(* IEC 61131-3 sources: digital-academy-template/src, 23 files *)

(* ---- Tipi.st ---- *)
NAMESPACE tipi

    TYPE  stato : (stop, forward, backward, unknown, error);
    END_TYPE

    TYPE
        colore : USINT (
            Undefined := USINT#0, // il pacco va nel magazzino "scarto feed"
            Red       := USINT#1,
            Orange    := USINT#2,
            Yellow    := USINT#3,
            Green     := USINT#4,
            Blue      := USINT#5,
            Indigo    := USINT#6,
            Violet    := USINT#7
        ) := Undefined;
    END_TYPE

    TYPE InventoryMode:
        (Fill, Empty);
    END_TYPE

END_NAMESPACE

(* ---- tipi.st ---- *)
NAMESPACE tipi

    TYPE  stato : (stop, forward, backward, unknown, error);
    END_TYPE

END_NAMESPACE

(* ---- function.st ---- *)
NAMESPACE Libreria

    FUNCTION  SelectSensorInput : USINT
        VAR_INPUT
            uIndex : USINT;
            in1 : USINT;
            in2 : USINT;
            in3 : USINT;
            in4 : USINT;
            in5 : USINT;
        END_VAR
        CASE uIndex OF
            USINT#0 : SelectSensorInput:= in1;
            USINT#1 : SelectSensorInput:= in2;
            USINT#2 : SelectSensorInput:= in3;
            USINT#3 : SelectSensorInput:= in4;
            USINT#4 : SelectSensorInput:= in5;
        END_CASE;
    END_FUNCTION
 END_NAMESPACE

(* ---- nonusato_function.st ---- *)
NAMESPACE Libreria

    FUNCTION  SelectSensorInput : USINT
        VAR_INPUT
            uIndex : USINT;
            in1 : USINT;
            in2 : USINT;
            in3 : USINT;
            in4 : USINT;
            in5 : USINT;
        END_VAR
        CASE uIndex OF
            USINT#0 : SelectSensorInput:= in1;
            USINT#1 : SelectSensorInput:= in2;
            USINT#2 : SelectSensorInput:= in3;
            USINT#3 : SelectSensorInput:= in4;
            USINT#4 : SelectSensorInput:= in5;
        END_CASE;
    END_FUNCTION
 END_NAMESPACE

(* ---- nonusato_Simulazione.st ---- *)
USING tipi;
USING System.Timer;
USING tempo;

NAMESPACE Libreria

    FUNCTION Simulazione

        VAR_INPUT
            Qnf : BOOL;
            Qdf : BOOL;
            Qtf : BOOL;
            Qn2 : BOOL;
            Qd2 : BOOL;
            Qt2 : BOOL;
            Qn3 : BOOL;
            Qd3 : BOOL;
            Qt3 : BOOL;
            Qn4 : BOOL;
            Qd4 : BOOL;
            Qt4 : BOOL;
            Qnc : BOOL;
            Qdc : BOOL;
            Qtc : BOOL;
        END_VAR

        VAR_OUTPUT
            Idf : USINT;
            Iff : BOOL := TRUE;
            Isf : BOOL;
            Imf : BOOL;
            Id2 : USINT;
            If2 : BOOL;
            Is2 : BOOL;
            Im2 : BOOL;
            Id3 : USINT;
            If3 : BOOL;
            Is3 : BOOL;
            Im3 : BOOL;
            Id4 : USINT;
            If4 : BOOL;
            Is4 : BOOL;
            Im4 : BOOL;
            Idc : USINT;
            Ifc : BOOL;
            Isc : BOOL;
            Imc : BOOL;
        END_VAR

        VAR_EXTERNAL
            elapsedtimer : tempo.Timer;
        END_VAR

        VAR
            tStopMotor : Time;//tempo movimento motori
        END_VAR

        //BLOCCO FEED
        IF Qnf AND Iff THEN //IF nastro principale feed va avanti AND pacco presente su nastro principale feed
            IF elapsedtimer.Check(Qnf,tStopMotor) THEN //TIMER DA SISTEMARE
                Iff := FALSE; //spegni fotocellula nastro principare feed
                Isf := TRUE; //accendi sensore pacco prima del deviatore feed
                //Idf := ... ; //il sensore riceve il colore del pacco
            END_IF;
        END_IF;

        IF Qdf AND Isf THEN //IF deviatore feed chiuso (sta deviando) AND pacco presente prima del deviatore feed
            //NB: il main attualmente non cambia i valori nel vettore Qd
            Isf := FALSE; //spegni sensore pacco prima del deviatore feed
            Imf := TRUE; //accendi fotocellula nastromagazzino feed
            IF Qtf AND elapsedtimer.Check(Imf,tStopMotor) THEN //IF nastro magazzino feed va avanti AND tempo passato
                Imf := FALSE;
            END_IF; //il pacco è arrivato al magazzino feed
        END_IF;

        //BLOCCO 2
        IF Qn2 AND If2 THEN //IF nastro principale va avanti AND pacco presente su nastro principale
            IF elapsedtimer.Check(Qnf,tStopMotor) THEN //TIMER DA SISTEMARE
                If2 := FALSE; //spegni fotocellula nastro principale
                Is2 := TRUE; //accendi sensore pacco prima del deviatore
                //Id2 := ... ; //il sensore riceve il colore del pacco
            END_IF;
        END_IF;

        IF Qd2 AND Is2 THEN //IF deviatore chiuso (sta deviando) AND pacco presente prima del deviatore
            //NB: il main attualmente non cambia i valori nel vettore Qd
            Is2 := FALSE; //spegni sensore pacco prima del deviatore
            Im2 := TRUE; //accendi fotocellula nastro magazzino
            IF Qt2 AND elapsedtimer.Check(Imf,tStopMotor) THEN //IF nastro magazzino va avanti AND tempo passato
                Im2 := FALSE;
            END_IF; //il pacco è arrivato al magazzino
        END_IF;

        //BLOCCO 3
        IF Qn3 AND If3 THEN //IF nastro principale va avanti AND pacco presente su nastro principale
            IF elapsedtimer.Check(Qnf,tStopMotor) THEN //TIMER DA SISTEMARE
                If3 := FALSE; //spegni fotocellula nastro principale
                Is3 := TRUE; //accendi sensore pacco prima del deviatore
                //Id3 := ... ; //il sensore riceve il colore del pacco
            END_IF;
        END_IF;

        IF Qd3 AND Is3 THEN //IF deviatore chiuso (sta deviando) AND pacco presente prima del deviatore
            //NB: il main attualmente non cambia i valori nel vettore Qd
            Is3 := FALSE; //spegni sensore pacco prima del deviatore
            Im3 := TRUE; //accendi fotocellula nastro magazzino feed
            IF Qt3 AND elapsedtimer.Check(Imf,tStopMotor) THEN //IF nastro magazzino va avanti AND tempo passato
                Im3 := FALSE;
            END_IF; //il pacco è arrivato al magazzino
        END_IF;

        //BLOCCO 4
        IF Qn4 AND If4 THEN //IF nastro principale va avanti AND pacco presente su nastro principale
            IF elapsedtimer.Check(Qnf,tStopMotor) THEN //TIMER DA SISTEMARE
                If4 := FALSE; //spegni fotocellula nastro principale
                Is4 := TRUE; //accendi sensore pacco prima del deviatore
                //Id4 := ... ; //il sensore riceve il colore del pacco
            END_IF;
        END_IF;

        IF Qd4 AND Is4 THEN //IF deviatore chiuso (sta deviando) AND pacco presente prima del deviatore
            //NB: il main attualmente non cambia i valori nel vettore Qd
            Is4 := FALSE; //spegni sensore pacco prima del deviatore
            Im4 := TRUE; //accendi fotocellula nastromagazzino
            IF Qt4 AND elapsedtimer.Check(Imf,tStopMotor) THEN //IF nastro magazzino va avanti AND tempo passato
                Im4 := FALSE;
            END_IF; //il pacco è arrivato al magazzino
        END_IF;

        //BLOCCO CODA
        IF Qnc AND Ifc THEN //IF nastro principale va avanti AND pacco presente su nastro principale
            IF elapsedtimer.Check(Qnf,tStopMotor) THEN //TIMER DA SISTEMARE
                Ifc := FALSE; //spegni fotocellula nastro principale
                Isc := TRUE; //accendi sensore pacco prima del deviatore
                //Idc := ... ; //il sensore riceve il colore del pacco
            END_IF;
        END_IF;

        IF Qdc AND Isc THEN //IF deviatore chiuso (sta deviando) AND pacco presente prima del deviatore
            //NB: il main attualmente non cambia i valori nel vettore Qd
            Isc := FALSE; //spegni sensore pacco prima del deviatore
            Imc := TRUE; //accendi fotocellula nastromagazzino
            IF Qtc AND elapsedtimer.Check(Imf,tStopMotor) THEN //IF nastro magazzino va avanti AND tempo passato
                Imc := FALSE;
            END_IF; //il pacco è arrivato al magazzino
        END_IF;

    END_FUNCTION

END_NAMESPACE

(* ---- SelectSensorInput.st ---- *)
NAMESPACE Libreria

    FUNCTION  SelectSensorInput : USINT
        VAR_INPUT
            uIndex : INT;
            in1 : USINT; //sensore colore deviatore nastro feed
            in2 : USINT; //sensore colore deviatore magazzino 2
            in3 : USINT; //sensore colore deviatore magazzino 3
            in4 : USINT; //sensore colore deviatore magazzino 4
            in5 : USINT; //sensore colore deviatore magazzino coda
        END_VAR
        CASE uIndex OF
            INT#1 : SelectSensorInput:= in1;
            INT#2 : SelectSensorInput:= in2;
            INT#3 : SelectSensorInput:= in3;
            INT#4 : SelectSensorInput:= in4;
            INT#5 : SelectSensorInput:= in5;
        END_CASE;
    END_FUNCTION
 END_NAMESPACE

(* ---- Simulazione.st ---- *)
//NOT WORKING PROPERLY AND NOT USED

USING tipi;
USING System.Timer;
USING tempo;

NAMESPACE Libreria

    FUNCTION Simulazione

        VAR_INPUT
            Qnf : BOOL;
            Qdf : BOOL;
            Qtf : BOOL;
            Qn2 : BOOL;
            Qd2 : BOOL;
            Qt2 : BOOL;
            Qn3 : BOOL;
            Qd3 : BOOL;
            Qt3 : BOOL;
            Qn4 : BOOL;
            Qd4 : BOOL;
            Qt4 : BOOL;
            Qnc : BOOL;
            Qdc : BOOL;
            Qtc : BOOL;
        END_VAR

        VAR_OUTPUT
            Idf : USINT;
            Iff : BOOL := TRUE;
            Isf : BOOL;
            Imf : BOOL;
            Id2 : USINT;
            If2 : BOOL;
            Is2 : BOOL;
            Im2 : BOOL;
            Id3 : USINT;
            If3 : BOOL;
            Is3 : BOOL;
            Im3 : BOOL;
            Id4 : USINT;
            If4 : BOOL;
            Is4 : BOOL;
            Im4 : BOOL;
            Idc : USINT;
            Ifc : BOOL;
            Isc : BOOL;
            Imc : BOOL;
        END_VAR

        VAR_EXTERNAL
            elapsedtimer : tempo.Timer;
        END_VAR

        VAR
            tStopMotor : Time;//tempo movimento motori
        END_VAR

        //BLOCCO FEED
        IF Qnf AND Iff THEN //IF nastro principale feed va avanti AND pacco presente su nastro principale feed
            IF elapsedtimer.Check(Qnf,tStopMotor) THEN //TIMER DA SISTEMARE
                Iff := FALSE; //spegni fotocellula nastro principare feed
                Isf := TRUE; //accendi sensore pacco prima del deviatore feed
                //Idf := ... ; //il sensore riceve il colore del pacco
            END_IF;
        END_IF;

        IF Qdf AND Isf THEN //IF deviatore feed chiuso (sta deviando) AND pacco presente prima del deviatore feed
            //NB: il main attualmente non cambia i valori nel vettore Qd
            Isf := FALSE; //spegni sensore pacco prima del deviatore feed
            Imf := TRUE; //accendi fotocellula nastromagazzino feed
            IF Qtf AND elapsedtimer.Check(Imf,tStopMotor) THEN //IF nastro magazzino feed va avanti AND tempo passato
                Imf := FALSE;
            END_IF; //il pacco è arrivato al magazzino feed
        END_IF;

        //BLOCCO 2
        IF Qn2 AND If2 THEN //IF nastro principale va avanti AND pacco presente su nastro principale
            IF elapsedtimer.Check(Qnf,tStopMotor) THEN //TIMER DA SISTEMARE
                If2 := FALSE; //spegni fotocellula nastro principale
                Is2 := TRUE; //accendi sensore pacco prima del deviatore
                //Id2 := ... ; //il sensore riceve il colore del pacco
            END_IF;
        END_IF;

        IF Qd2 AND Is2 THEN //IF deviatore chiuso (sta deviando) AND pacco presente prima del deviatore
            //NB: il main attualmente non cambia i valori nel vettore Qd
            Is2 := FALSE; //spegni sensore pacco prima del deviatore
            Im2 := TRUE; //accendi fotocellula nastro magazzino
            IF Qt2 AND elapsedtimer.Check(Imf,tStopMotor) THEN //IF nastro magazzino va avanti AND tempo passato
                Im2 := FALSE;
            END_IF; //il pacco è arrivato al magazzino
        END_IF;

        //BLOCCO 3
        IF Qn3 AND If3 THEN //IF nastro principale va avanti AND pacco presente su nastro principale
            IF elapsedtimer.Check(Qnf,tStopMotor) THEN //TIMER DA SISTEMARE
                If3 := FALSE; //spegni fotocellula nastro principale
                Is3 := TRUE; //accendi sensore pacco prima del deviatore
                //Id3 := ... ; //il sensore riceve il colore del pacco
            END_IF;
        END_IF;

        IF Qd3 AND Is3 THEN //IF deviatore chiuso (sta deviando) AND pacco presente prima del deviatore
            //NB: il main attualmente non cambia i valori nel vettore Qd
            Is3 := FALSE; //spegni sensore pacco prima del deviatore
            Im3 := TRUE; //accendi fotocellula nastro magazzino feed
            IF Qt3 AND elapsedtimer.Check(Imf,tStopMotor) THEN //IF nastro magazzino va avanti AND tempo passato
                Im3 := FALSE;
            END_IF; //il pacco è arrivato al magazzino
        END_IF;

        //BLOCCO 4
        IF Qn4 AND If4 THEN //IF nastro principale va avanti AND pacco presente su nastro principale
            IF elapsedtimer.Check(Qnf,tStopMotor) THEN //TIMER DA SISTEMARE
                If4 := FALSE; //spegni fotocellula nastro principale
                Is4 := TRUE; //accendi sensore pacco prima del deviatore
                //Id4 := ... ; //il sensore riceve il colore del pacco
            END_IF;
        END_IF;

        IF Qd4 AND Is4 THEN //IF deviatore chiuso (sta deviando) AND pacco presente prima del deviatore
            //NB: il main attualmente non cambia i valori nel vettore Qd
            Is4 := FALSE; //spegni sensore pacco prima del deviatore
            Im4 := TRUE; //accendi fotocellula nastromagazzino
            IF Qt4 AND elapsedtimer.Check(Imf,tStopMotor) THEN //IF nastro magazzino va avanti AND tempo passato
                Im4 := FALSE;
            END_IF; //il pacco è arrivato al magazzino
        END_IF;

        //BLOCCO CODA
        IF Qnc AND Ifc THEN //IF nastro principale va avanti AND pacco presente su nastro principale
            IF elapsedtimer.Check(Qnf,tStopMotor) THEN //TIMER DA SISTEMARE
                Ifc := FALSE; //spegni fotocellula nastro principale
                Isc := TRUE; //accendi sensore pacco prima del deviatore
                //Idc := ... ; //il sensore riceve il colore del pacco
            END_IF;
        END_IF;

        IF Qdc AND Isc THEN //IF deviatore chiuso (sta deviando) AND pacco presente prima del deviatore
            //NB: il main attualmente non cambia i valori nel vettore Qd
            Isc := FALSE; //spegni sensore pacco prima del deviatore
            Imc := TRUE; //accendi fotocellula nastromagazzino
            IF Qtc AND elapsedtimer.Check(Imf,tStopMotor) THEN //IF nastro magazzino va avanti AND tempo passato
                Imc := FALSE;
            END_IF; //il pacco è arrivato al magazzino
        END_IF;

    END_FUNCTION

END_NAMESPACE

(* ---- Tempo.st ---- *)
FUNCTION Timer: BOOL
    VAR_INPUT
        tStopMotor: INT;   // Tempo massimo che la funzione aspetta
    END_VAR

    VAR
        tTemp: INT := 0;   // Variabile temporanea per il conteggio
    END_VAR

    Timer:=FALSE;
    // Ciclo WHILE per incrementare il valore di t fino a tStopMotor
    WHILE tTemp < tStopMotor DO
        tTemp := tTemp + 1;
    END_WHILE;

    // Dopo aver completato il ciclo, ritorna TRUE (indica che è finito)
    Timer := TRUE;

END_FUNCTION

(* ---- Deviatore.st ---- *)
USING Tipi;

NAMESPACE Libreria

    CLASS deviatore

        VAR PUBLIC
            ID :INT;
            color : colore;
            sensore : BOOL; // il sensore del deviatore del magazzino rosso si attiva se vede un pacco rosso
            cntrlApri : BOOL; // segnale per aprire il deviatore (se è aperto lascia passare i pacchi)
            cntrlChiudi : BOOL; // segnale per chiudere il deviatore (se è chiuso devia i pacchi)
            chiuso : BOOL;
            accetta : BOOL;
        END_VAR

        METHOD PUBLIC Init // inizializzazione del deviatore
            VAR_INPUT
                IDinit : INT;
            END_VAR
            ID:=IDinit;
            sensore := FALSE; // all'inizio non vede il pacco
            chiuso := FALSE; // all'inizio il deviatore è aperto
            cntrlApri := FALSE;
            cntrlChiudi := FALSE; // all'inizio non ci sono comandi di apertura o chiusura
        END_METHOD

        METHOD PUBLIC ChiudiDeviatore : BOOL // nel main se (sensore = TRUE) vogliamo chiudere il deviatore

            cntrlChiudi := TRUE;

        END_METHOD

        METHOD PUBLIC ApriDeviatore : BOOL // una volta deviato il pacco nel mai (sensore = FALSE) vogliamo aprire il deviatore
            cntrlApri := TRUE;
            cntrlChiudi := FALSE;
            chiuso := FALSE;
        END_METHOD // NB ci pensa test.st a definire (chiuso := FALSE)

        METHOD PUBLIC Accept

            cntrlChiudi := TRUE;

        END_METHOD

        METHOD PUBLIC Discard : BOOL

            cntrlApri := TRUE;

        END_METHOD

        METHOD PUBLIC IsMyColor : BOOL  //controlla se accettare o meno il pacco
            VAR_INPUT
                uSensor:colore;
            END_VAR

            IF uSensor = color THEN
                IsMyColor := TRUE;
            ELSE
                IsMyColor := FALSE;
            END_IF;

        END_METHOD

    END_CLASS

END_NAMESPACE

(* ---- deviatore.st ---- *)
USING Tipi;

NAMESPACE Libreria

    CLASS deviatore

        VAR PUBLIC
            ID :INT;
            sensore : BOOL; // il sensore del deviatore del magazzino rosso si attiva se vede un pacco rosso
            cntrlApri : BOOL; // segnale per aprire il deviatore (se è aperto lascia passare i pacchi)
            cntrlChiudi : BOOL; // segnale per chiudere il deviatore (se è chiuso devia i pacchi)
            chiuso : BOOL;
        END_VAR

        METHOD PUBLIC Init // inizializzazione del deviatore
            VAR_INPUT
                IDinit : INT;
            END_VAR
            ID:=IDinit;
            sensore := FALSE; // all'inizio non vede il pacco
            chiuso := FALSE; // all'inizio il deviatore è aperto
            cntrlApri := FALSE;
            cntrlChiudi := FALSE; // all'inizio non ci sono comandi di apertura o chiusura
        END_METHOD

        METHOD PUBLIC ChiudiDeviatore // nel main se (sensore = TRUE) vogliamo chiudere il deviatore
            cntrlChiudi := TRUE;
            cntrlApri := FALSE;
        END_METHOD // NB ci pensa test.st a definire (chiuso := TRUE)

        METHOD PUBLIC ApriDeviatore // una volta deviato il pacco nel mai (sensore = FALSE) vogliamo aprire il deviatore
            cntrlApri := TRUE;
            cntrlChiudi := FALSE;
        END_METHOD // NB ci pensa test.st a definire (chiuso := FALSE)

    END_CLASS

END_NAMESPACE

(* ---- Inventory.st ---- *)
USING Tipi;
USING Libreria;

NAMESPACE Libreria

    CLASS PUBLIC Inventory EXTENDS nastro
        VAR PUBLIC
            IDpackage: INT;
            ListStoredPackages: ARRAY[1..100] OF USINT; //dato che un magazzino deve avere pacchi dello stesso colore, può servire per controllare che tutti i pacchi inseriti abbiano effettivamente lo stesso colore
            currentStockLevel: INT; //livello di stock attuale
            maxCapacity: INT; //capacità massima
            acceptedColor: USINT;
            StockisFull: BOOL;
            currentMode: Tipi.InventoryMode;
            statomotore: stato;
            recipe: Ricetta;
        END_VAR

        METHOD PUBLIC Init //initialization of the inventory
            VAR_INPUT
                Capacity : INT;
                Color : USINT;
                ID_i: INT;
            END_VAR
            maxCapacity := Capacity;
            acceptedColor := Color;
            IDpackage:= ID_i;
            currentStockLevel:=0; //ipotizzo che inizialmente i magazzini siano vuoti
            StockisFull := FALSE;
            currentMode := Tipi.InventoryMode#Fill; // di default vogliamo riempire i magazzini
        END_METHOD

        METHOD PUBLIC isFull  //controlla se il magazzino è pieno
            VAR_OUTPUT
                Load: BOOL; //TRUE:"ok puoi ancora riempire", FALSE:non puoi riempire
            END_VAR

            IF currentStockLevel < maxCapacity THEN
                StockisFull:= FALSE;
                Load:=TRUE;
            ELSE
                StockisFull:=TRUE;
                Load:=FALSE;
            END_IF;
        END_METHOD

        METHOD PUBLIC GetCurrentStockLevel : INT  //se chiamato, mostra il livello di riempimento attuale
            GetCurrentStockLevel:= currentStockLevel;
        END_METHOD

        METHOD PUBLIC EmptyFIFO
            VAR
                i: INT;
            END_VAR

            FOR i := 1 TO currentStockLevel - 1 DO
                ListStoredPackages[i] := ListStoredPackages[i + 1]; // Shift dei pacchi a sinistra (FIFO)
            END_FOR;
            ListStoredPackages[currentStockLevel] := TO_USINT(0); //resetto l'ultima posizione
            currentStockLevel := currentStockLevel - 1;

            IF currentStockLevel = 0 THEN
                statomotore := Tipi.stato#stop;
                currentMode:=Tipi.InventoryMode#Fill;
            END_IF;
        END_METHOD

        METHOD PUBLIC SetMode // MODALITà RIEMPIMENTO O SVUOTAMENTO, LOGICA:FIFO
            VAR_INPUT
                mode : Tipi.InventoryMode;
                //InventorySensor:BOOL;
                InventoryPhotocell: BOOL; //c'è un pacco sul nastro del magazzino?
                DiverterSensor: BOOL; //se TRUE il deviatore è chiuso e manda il pacco al magazzino
                ID_i: USINT;
            END_VAR
            currentMode := mode;
            IF currentMode= InventoryMode#Fill THEN
                IF StockisFull=FALSE AND DiverterSensor=TRUE AND statomotore=Tipi.stato#forward AND InventoryPhotocell=TRUE THEN
                    currentStockLevel:=currentStockLevel+1;
                    ListStoredPackages[currentStockLevel]:= ID_i; //salvo l'ID_i del pacco n nell'n-esima posizione dell'array
                ELSIF StockisFull=TRUE THEN
                    RETURN; //magari inserire una variabile tipo warningCode/exitflag...
                END_IF;
            ELSE // the mode is set to "empty"
                IF recipe.RecipeSatisfiable()=TRUE THEN //AND currentStockLevel > 0 THEN
                    statomotore := Tipi.stato#backward;
                    THIS.EmptyFIFO();
                END_IF;
            END_IF;
        END_METHOD

    END_CLASS

END_NAMESPACE

(* ---- inventory.st ---- *)
USING Tipi;

NAMESPACE Inventory_lib

    CLASS PUBLIC Inventory
        VAR PUBLIC
            IDpackage: INT;
            ListStoredPackages: ARRAY[1..100] OF USINT; //dato che un magazzino deve avere pacchi dello stesso colore, può servire per controllare che tutti i pacchi inseriti abbiano effettivamente lo stesso colore
            currentStockLevel: INT; //livello di stock attuale
            maxCapacity: INT; //capacità massima
            acceptedColor: USINT;
            StockisFull: BOOL;
            currentMode: Tipi.InventoryMode;
        END_VAR

        METHOD PUBLIC Init //initialization of the inventory
            VAR_INPUT
                Capacity : INT;
                Color : USINT; //oppure tipi.colore#... oppure semplicemente INT e lo legge da solo?
                ID: INT;
            END_VAR
            maxCapacity := Capacity;
            acceptedColor := Color;
            IDpackage:= ID; //anche qui sarebbe color... forse non ha senso avere sia color che ID
            currentStockLevel:=0; //ipotizzo che inizialmente i magazzini siano vuoti
            StockisFull:=FALSE;
            currentMode := Tipi.InventoryMode#Fill; // di default vogliamo riempire i magazzini
        END_METHOD

        METHOD PUBLIC isFull  //controlla se il magazzino è pieno
            VAR_OUTPUT
                StockisFull: BOOL;
                Load: BOOL; //TRUE:"ok puoi ancora riempire", FALSE:non puoi riempire
            END_VAR
            IF currentStockLevel < maxCapacity THEN
                StockisFull:= FALSE;
                Load:=TRUE;
            ELSE
                StockisFull:=TRUE;
                Load:=FALSE;
            END_IF;
        END_METHOD

        METHOD PUBLIC GetCurrentStockLevel : INT  //se chiamato, mostra il livello di riempimento attuale
            GetCurrentStockLevel:= currentStockLevel;
        END_METHOD

        METHOD PUBLIC SetMode // MODALITà RIEMPIMENTO O SVUOTAMENTO, LOGICA:FIFO
            VAR_INPUT
                mode : Tipi.InventoryMode;
                //InventorySensor:BOOL;
                InventoryPhotocell: BOOL; //c'è un pacco sul nastro del magazzino?
                DiverterSensor: BOOL; //se TRUE il deviatore è chiuso e manda il pacco al magazzino
                ID: USINT;
            END_VAR
            currentMode := mode;
            IF currentMode= InventoryMode#Fill THEN
                IF StockisFull=FALSE AND DiverterSensor=TRUE AND Tipi.stato=Tipi.stato#forward AND InventoryPhotocell=TRUE THEN
                    currentStockLevel:=currentStockLevel+1;
                    ListStoredPackages[currentStockLevel]:= ID; //salvo l'ID del pacco n nell'n-esima posizione dell'array
                ELSIF StockisFull=TRUE THEN
                    RETURN; //magari inserire una variabile tipo warningCode/exitflag...
                END_IF;
            /*ELSE // the mode is set to "empty"
                IF RecipeSatisfiable=TRUE AND Tipi.stato=backward THEN
                    currentStockLevel:=currentStockLevel-;
                END_IF*///DA COMPLETARE
            END_IF;
        END_METHOD

    END_CLASS

END_NAMESPACE

/*{Test}
METHOD PUBLIC MyTestMethod
    ; // AxUnit.Assert.Equal(y, x)
END_METHOD*/

(* ---- Magazzino.st ---- *)
USING Tipi;

NAMESPACE Libreria

    CLASS magazzino

        VAR PUBLIC
            ID:INT;
            isFull: BOOL;
            colore : colore;
            i:INT;
            spazio:INT;
            fotocellula:BOOL;
            actualState : stato;
            CntrlForward : BOOL;    // Comando avanti
            CntrlBackward : BOOL;   // Comando indietro
            isForward : BOOL;    // Uscita avanti
            isBackward : BOOL;   // Uscita indietro

        END_VAR

        METHOD PUBLIC Init  // Init motor
            VAR_INPUT
                IDinit : INT;
                Color : colore;
            END_VAR
            ID:=IDinit;
            colore := color;
            actualState := stato#stop;
            CntrlForward := FALSE;
            CntrlBackward := FALSE;
            isForward := FALSE;
            isBackward := FALSE;

        END_METHOD

        METHOD PUBLIC Update

            IF CntrlForward AND NOT CntrlBackward THEN
                actualState := stato#forward;
            ELSIF CntrlBackward AND NOT CntrlForward THEN
                actualState := stato#backward;
            ELSE
                actualState := stato#stop;
            END_IF;

            CASE actualState OF
                stato#forward:
                    isForward := TRUE;
                    isBackward := FALSE;
                stato#backward:
                    isForward := FALSE;
                    isBackward := TRUE;
                stato#stop:
                    isForward := FALSE;
                    isBackward := FALSE;
            END_CASE;
            END_METHOD

    END_CLASS

END_NAMESPACE

(* ---- magazzino.st ---- *)
USING Tipi;

NAMESPACE Libreria

    CLASS magazzino

        VAR PUBLIC
            ID:INT;
            isFull: BOOL;
            colore : colore;
            i:INT;
            spazio:INT;
            sensore:BOOL;
            actualState : stato;
            CntrlForward : BOOL;    // Comando avanti
            CntrlBackward : BOOL;   // Comando indietro
            isForward : BOOL;    // Uscita avanti
            isBackward : BOOL;   // Uscita indietro

        END_VAR

        METHOD PUBLIC Init  // Init motor
            VAR_INPUT
                IDinit : INT;
            END_VAR
            ID:=IDinit;
            colore := colore;
            actualState := stato#stop;
            CntrlForward := FALSE;
            CntrlBackward := FALSE;
            isForward := FALSE;
            isBackward := FALSE;

        END_METHOD

        METHOD PUBLIC Update

            IF CntrlForward AND NOT CntrlBackward THEN
                actualState := stato#forward;
            ELSIF CntrlBackward AND NOT CntrlForward THEN
                actualState := stato#backward;
            ELSE
                actualState := stato#stop;
            END_IF;

            CASE actualState OF
                stato#forward:
                    isForward := TRUE;
                    isBackward := FALSE;
                stato#backward:
                    isForward := FALSE;
                    isBackward := TRUE;
                stato#stop:
                    isForward := FALSE;
                    isBackward := FALSE;
            END_CASE;
            END_METHOD

    END_CLASS

END_NAMESPACE

(* ---- Nastro.st ---- *)
USING tipi;
//USING MotorClass; //preso da libreria di @sara_vecchio

NAMESPACE Libreria

    CLASS nastro

        VAR PUBLIC
            ID:INT;
            actualState : stato;    // Comando avanti
            CntrlBackward : BOOL;   // Comando indietro
            isForward : BOOL;    // Uscita avanti //necessario?
            isBackward : BOOL;   // Uscita indietro //necessario?
            isEmpty:BOOL;
            CntrlForward : BOOL;
            colore: colore;
        END_VAR

        METHOD PUBLIC Init  // Initialization motor
            VAR_INPUT
                IDinit : INT;
                Color : colore;
            END_VAR
            ID:=IDinit;
            colore := color;
            actualState := stato#stop;
            CntrlForward := FALSE;
            CntrlBackward := FALSE;
            isForward := FALSE;
            isBackward := FALSE;

        END_METHOD

        METHOD PUBLIC Update : stato

            IF CntrlForward AND NOT CntrlBackward THEN
                actualState := stato#forward;
            ELSIF CntrlBackward AND NOT CntrlForward THEN
                actualState := stato#backward;
            ELSE
                actualState := stato#stop;
            END_IF;

            CASE actualState OF
                stato#forward:
                    isForward := TRUE;
                    isBackward := FALSE;
                stato#backward:
                    isForward := FALSE;
                    isBackward := TRUE;
                stato#stop:
                    isForward := FALSE;
                    isBackward := FALSE;
            END_CASE;

        END_METHOD

        METHOD PUBLIC CheckEmpty : BOOL  //check if is isEmpty from sensor

            VAR_INPUT
                bLightSensor: BOOL;
            END_VAR

            IF bLightSensor THEN
                CheckEmpty := FALSE;
            ELSIF NOT bLightSensor THEN
                CheckEmpty := TRUE;
            ELSE
                actualState := stato#error;
            END_IF;

        END_METHOD

        METHOD PUBLIC GetStatus : tipi.stato // get state of the conveyor
            GetStatus := actualState;
        END_METHOD

        METHOD PUBLIC Stop : BOOL
            CntrlForward := FALSE;
            CntrlBackward := FALSE;
            actualState := stato#stop;
            //Stop:=????
        END_METHOD

        METHOD PUBLIC RunForward : BOOL //serve chiamare anche i motori?
            IF actualState <> stato#error THEN
                //Motor.Start := TRUE;
                CntrlForward := TRUE; //aggiungi sicura per eviatre che avanti e indietro possano essere attivati contemporaneamente
                actualState := stato#forward;
            END_IF;
            RunForward:=CntrlForward;
        END_METHOD

        METHOD PUBLIC RunBackward
            IF actualState <> stato#error THEN
                //Motor.Start := TRUE;
                CntrlBackward := TRUE; //aggiungi stessa sicura di sopra
                actualState := stato#backward;
            END_IF;
        END_METHOD

    END_CLASS

END_NAMESPACE

(* ---- nastro.st ---- *)
USING Tipi;

NAMESPACE Libreria

    CLASS nastro

        VAR PUBLIC
            ID:INT;
            isEmpty: BOOL;
            actualState : stato;
            CntrlForward : BOOL;    // Comando avanti
            CntrlBackward : BOOL;   // Comando indietro
            isForward : BOOL;    // Uscita avanti
            isBackward : BOOL;   // Uscita indietro
            i:INT;
        END_VAR

        METHOD PUBLIC Init  // Init motor
            VAR_INPUT
                IDinit : INT;
            END_VAR
            ID:=IDinit;
            actualState := stato#stop;
            CntrlForward := FALSE;
            CntrlBackward := FALSE;
            isForward := FALSE;
            isBackward := FALSE;

        END_METHOD

        METHOD PUBLIC Update

            IF CntrlForward AND NOT CntrlBackward THEN
                actualState := stato#forward;
            ELSIF CntrlBackward AND NOT CntrlForward THEN
                actualState := stato#backward;
            ELSE
                actualState := stato#stop;
            END_IF;

            CASE actualState OF
                stato#forward:
                    isForward := TRUE;
                    isBackward := FALSE;
                stato#backward:
                    isForward := FALSE;
                    isBackward := TRUE;
                stato#stop:
                    isForward := FALSE;
                    isBackward := FALSE;
            END_CASE;

        END_METHOD

        METHOD PUBLIC fotocellula  //check if is isEmpty from sensor
                isEmpty := TRUE;
        END_METHOD

        METHOD PUBLIC GetStatus // get state of the conveyor
            actualState:=actualState;
        END_METHOD
    END_CLASS

END_NAMESPACE

(* ---- nonusato_Ricetta.st ---- *)
USING tipi;

NAMESPACE Libreria

    CLASS PUBLIC Ricetta

        /*STRUCT RicettaTipo
            Colore: USINT; // colore desiderato
            Quantità: INT; // numero pacchi necessari
        END_STRUCT

        VAR_GLOBAL
            Ricetta : ARRAY[1..5] OF RicettaTipo; // max 5 tipi di pacchi richiesti
        END_VAR*/

        METHOD PUBLIC RecipeSatisfiable : BOOL
            VAR
                i: INT;
                matchingColor: USINT;
                matchingQuantity: INT;
                foundCount: INT;
            END_VAR

            RecipeSatisfiable := TRUE; // assumi che sia soddisfatta, fino a prova contraria

            /*FOR i := 1 TO SIZEOF(Tipi.Ricetta) DO
                matchingColor := Tipi.Ricetta[i].Colore;
                matchingQuantity := Tipi.Ricetta[i].Quantità;

                // Verifica se il magazzino ha il colore richiesto
                IF acceptedColor = matchingColor THEN
                    IF currentStockLevel < matchingQuantity THEN
                        RecipeSatisfiable := FALSE;
                        RETURN;
                    END_IF;
                END_IF;
            END_FOR;*/

        END_METHOD

        /*METHOD PUBLIC RecipeSatisfiable:BOOL
            IF Ricetta.HowMany THEN
                RecipeSatisfiable:=TRUE;
            ELSE
                RecipeSatisfiable:=FALSE;
            END_IF;
        END_METHOD*/

    END_CLASS

END_NAMESPACE

(* ---- nonusato_Tempo.st ---- *)
USING System.Timer;

NAMESPACE tempo

    Class Timer

    VAR
        ton : OnDelay;
    END_VAR

    METHOD PUBLIC Check : BOOL
        VAR_INPUT
            signal: BOOL;
            duration : time;
            timeout : time;
        END_VAR
        ton(signal := TRUE, duration := Timeout);
        IF (ton.output) THEN
            Check := TRUE;
        ELSE
           Check := FALSE;
        END_IF;
    END_METHOD

    METHOD PUBLIC Reset
        ton(signal:= FALSE);
    END_METHOD

    END_class

END_NAMESPACE

(* ---- Ricetta.st ---- *)
//TO BE COMPLETED; NOT USED YET

USING tipi;

NAMESPACE Libreria

    CLASS PUBLIC Ricetta

        /*STRUCT RicettaTipo
            Colore: USINT; // colore desiderato
            Quantità: INT; // numero pacchi necessari
        END_STRUCT

        VAR_GLOBAL
            Ricetta : ARRAY[1..5] OF RicettaTipo; // max 5 tipi di pacchi richiesti
        END_VAR*/

        METHOD PUBLIC RecipeSatisfiable : BOOL
            VAR
                i: INT;
                matchingColor: USINT;
                matchingQuantity: INT;
                foundCount: INT;
            END_VAR

            RecipeSatisfiable := TRUE; // assumi che sia soddisfatta, fino a prova contraria

            /*FOR i := 1 TO SIZEOF(Tipi.Ricetta) DO
                matchingColor := Tipi.Ricetta[i].Colore;
                matchingQuantity := Tipi.Ricetta[i].Quantità;

                // Verifica se il magazzino ha il colore richiesto
                IF acceptedColor = matchingColor THEN
                    IF currentStockLevel < matchingQuantity THEN
                        RecipeSatisfiable := FALSE;
                        RETURN;
                    END_IF;
                END_IF;
            END_FOR;*/

        END_METHOD

        /*METHOD PUBLIC RecipeSatisfiable:BOOL
            IF Ricetta.HowMany THEN
                RecipeSatisfiable:=TRUE;
            ELSE
                RecipeSatisfiable:=FALSE;
            END_IF;
        END_METHOD*/

    END_CLASS

END_NAMESPACE

(* ---- Configuration.st ---- *)
USING Siemens.Simatic.S71500.Tasks;
USING tipi;
USING Libreria;

CONFIGURATION MyConfig

    TASK Load: Startup;
    TASK Main(Interval := T#100ms,PRIORITY:=1); //di default è 50ms (minimo)

    PROGRAM P0 WITH Load: LoadConfiguration;
    PROGRAM P1 WITH Main: MainProgram;

    // Configuring IO tags
    VAR_GLOBAL

        //input output feed
        Qnf AT %Q0.0 : BOOL; //output nastro feed
        Qnc AT %Q0.1 : BOOL;
        Qn2 AT %Q0.2 : BOOL;
        Qn3 AT %Q0.3 : BOOL;
        Qn4 AT %Q0.4 : BOOL;

        Qdf AT %Q1.0 : BOOL; //output deviatore feed
        Qdc AT %Q1.1 : BOOL;
        Qd2 AT %Q1.2 : BOOL;
        Qd3 AT %Q1.3 : BOOL;
        Qd4 AT %Q1.4 : BOOL;

        Qtf AT %Q2.0 : BOOL; //output tank feed
        Qtc AT %Q2.1 : BOOL;
        Qt2 AT %Q2.2 : BOOL;
        Qt3 AT %Q2.3 : BOOL;
        Qt4 AT %Q2.4 : BOOL;

        Idf AT %IB6 : USINT; //input deviatore feed (colore)
        Idc AT %IB7 : USINT;
        Id2 AT %IB8 : USINT;
        Id3 AT %IB9 : USINT;
        Id4 AT %IB10 : USINT;

        Iff AT %I0.0 : BOOL; //input fotocellula feed (presenza pacco su nastro principale)
        Ifc AT %I0.1 : BOOL;
        If2 AT %I0.2 : BOOL;
        If3 AT %I0.3 : BOOL;
        If4 AT %I0.4 : BOOL;

        Isf AT %I1.0 : BOOL; //input sensore feed (presenza pacco su nastro principale prima del deviatore)
        Isc AT %I1.1 : BOOL;
        Is2 AT %I1.2 : BOOL;
        Is3 AT %I1.3 : BOOL;
        Is4 AT %I1.4 : BOOL;

        Imf AT %I2.0 : BOOL; //input magazzino feed (presenza pacco su nastro principale)
        Imc AT %I2.1 : BOOL;
        Im2 AT %I2.2 : BOOL;
        Im3 AT %I2.3 : BOOL;
        Im4 AT %I2.4 : BOOL;

    END_VAR

    VAR_GLOBAL

        nastri : ARRAY[1..n_mag] OF nastro;
        deviatori : ARRAY[1..n_mag] OF deviatore;
        magazzini : ARRAY[1..n_mag] OF inventory;

    END_VAR

    VAR_GLOBAL CONSTANT

        n_mag : INT := 5; // numero magazzini considerando uno feed e uno scarto e il penultimo ricetta o semplice
        capacity : INT := 20; //numero pacchi che ogni magazzino può contenere

    END_VAR

END_CONFIGURATION

PROGRAM LoadConfiguration

    VAR_EXTERNAL

        nastri : ARRAY [1..n_mag] OF Libreria.nastro;
        deviatori : ARRAY [1..n_mag] OF Libreria.deviatore;
        magazzini : ARRAY [1..n_mag] OF Libreria.inventory;

        Qnf : BOOL;
        Qdf : BOOL;
        Qtf : BOOL;
        Idf : USINT;
        Iff : BOOL;
        Isf : BOOL;
        Imf : BOOL;
        Qnc : BOOL;
        Qdc : BOOL;
        Qtc : BOOL;
        Idc : USINT;
        Ifc : BOOL;
        Isc : BOOL;
        Imc : BOOL;
        Qn2 : BOOL;
        Qd2 : BOOL;
        Qt2 : BOOL;
        Id2 : USINT;
        If2 : BOOL;
        Is2 : BOOL;
        Im2 : BOOL;
        Qn3 : BOOL;
        Qd3 : BOOL;
        Qt3 : BOOL;
        Id3 : USINT;
        If3 : BOOL;
        Is3 : BOOL;
        Im3 : BOOL;
        Qn4 : BOOL;
        Qd4 : BOOL;
        Qt4 : BOOL;
        Id4 : USINT;
        If4 : BOOL;
        Is4 : BOOL;
        Im4 : BOOL;

    END_VAR

    VAR_EXTERNAL CONSTANT
        n_mag : INT;
        capacity : INT;
    END_VAR

    //inizializzo il blocco feed
    nastri[1].Init(1);
    deviatori[1].Init(1, colore#Undefined); //qua dico anche che colore il deviatore deve accettare
    magazzini[1].Init_magazzino(1, capacity);

    //inizializzo il blocco 2
    nastri[2].Init(2);
    deviatori[2].Init(2, colore#Red); //qua dico anche che colore il deviatore deve accettare
    magazzini[2].Init_magazzino(2, capacity);

    //inizializzo il blocco 3
    nastri[3].Init(3);
    deviatori[3].Init(3, colore#White); //qua dico anche che colore il deviatore deve accettare
    magazzini[3].Init_magazzino(3, capacity);

    //inizializzo il blocco 4
    nastri[4].Init(4);
    deviatori[4].Init(4, colore#Yellow); //qua dico anche che colore il deviatore deve accettare
    magazzini[4].Init_magazzino(4, capacity);

    //inizializzo il blocco coda
    nastri[n_mag].Init(n_mag);
    deviatori[n_mag].Init(n_mag, colore#Undefined); //qua dico un colore a caso ma in realtà accetta tutto (vedi method deviatore.IsMyColor_coda)
    magazzini[n_mag].Init_magazzino(n_mag, capacity);

END_PROGRAM

(* ---- configuration.st ---- *)
CONFIGURATION MyConfiguration
    TASK Main(Priority := 1);

    PROGRAM P1 WITH Main: MainProgram;

    VAR_GLOBAL
        Tag1 : INT;
        Tag3 AT %IB4 : BYTE;
    END_VAR

    VAR_GLOBAL CONSTANT
        Tag2 : BOOL := TRUE ;
    END_VAR

END_CONFIGURATION

(* ---- LoadPlantConfiguration.st ---- *)
USING tipi;

PROGRAM LoadPlantConfiguration

    VAR_TEMP
        i:INT :=0;
    END_VAR

    VAR
    coloreq : USINT;
    END_VAR

    VAR_EXTERNAL
        nastri : ARRAY [1..n_mag] OF Libreria.nastro;
        deviatori : ARRAY [1..n_mag] OF Libreria.deviatore;
        magazzini : ARRAY [1..n_mag] OF Libreria.inventory;
        //Qn : REF_TO ARRAY[1..n_mag] of BOOL ;
        //Qd : ARRAY[1..n_mag] of BOOL ;
        //Qt : ARRAY[1..n_mag] of BOOL ;
        Id : ARRAY[1..n_mag] of USINT ;
        If_ : ARRAY[1..n_mag] of BOOL ;
        Is : ARRAY[1..n_mag] of BOOL ;
        Im : ARRAY[1..n_mag] of BOOL ;

        Qn: BYTE;
        Qd: BYTE;
        Qt: BYTE;
        //Id: BYTE;
    //    If_ :BYTE;
    //    Is:BYTE;
    //    Im:BYTE;

        Qnf : BOOL;
        Qdf : BOOL;
        Qtf : BOOL;
        Idf : USINT;
        Iff : BOOL;
        Isf : BOOL;
        Imf : BOOL;
        Qnc : BOOL;
        Qdc : BOOL;
        Qtc : BOOL;
        Idc : USINT;
        Ifc : BOOL;
        Isc : BOOL;
        Imc : BOOL;
        Qn2 : BOOL;
        Qd2 : BOOL;
        Qt2 : BOOL;
        Id2 : USINT;
        If2 : BOOL;
        Is2 : BOOL;
        Im2 : BOOL;
        Qn3 : BOOL;
        Qd3 : BOOL;
        Qt3 : BOOL;
        Id3 : USINT;
        If3 : BOOL;
        Is3 : BOOL;
        Im3 : BOOL;
        Qn4 : BOOL;
        Qd4 : BOOL;
        Qt4 : BOOL;
        Id4 : USINT;
        If4 : BOOL;
        Is4 : BOOL;
        Im4 : BOOL;
        //n_pacchi : INT;
        elapsedtimer : tempo.Timer;

    END_VAR

    VAR_EXTERNAL CONSTANT
        n_mag : INT;
        capacity : INT;
        n_pacchi : INT;
    END_VAR

        /*Qn[1]  := Qnf;
        Qn[2]  := Qn2;
        Qn[3]  := Qn3;
        Qn[4]  := Qn4;
        Qn[5]  := Qnc;

        Qd[1]  := Qdf;
        Qd[2]  := Qd2;
        Qd[3]  := Qd3;
        Qd[4]  := Qd4;
        Qd[5]  := Qdc;

        Qt[1]  := Qtf;
        Qt[2]  := Qt2;
        Qt[3]  := Qt3;
        Qt[4]  := Qt4;
        Qt[5]  := Qtc;*/

        Id[1]  := Idf;
        Id[2]  := Id2;
        Id[3]  := Id3;
        Id[4]  := Id4;
        Id[5]  := Idc;

        If_[1] := Iff;
        If_[2] := If2;
        If_[3] := If3;
        If_[4] := If4;
        If_[5] := Ifc;

        Is[1] := Isf;
        Is[2] := Is2;
        Is[3] := Is3;
        Is[4] := Is4;
        Is[5] := Isc;

        Im[1] := Imf;
        Im[2] := Im2;
        Im[3] := Im3;
        Im[4] := Im4;
        Im[5] := Imc;

        //feed
        nastri[1].ID := 1;
        nastri[1].colore := USINT#0;
        nastri[1].actualState := stato#stop;
        nastri[1].CntrlForward := FALSE;
        nastri[1].CntrlBackward := FALSE;
        nastri[1].isForward := FALSE;
        nastri[1].isBackward := FALSE;

        deviatori[1].ID:=nastri[1].ID;
        deviatori[1].sensore := FALSE;
        deviatori[1].chiuso := FALSE;
        deviatori[1].cntrlApri := FALSE;
        deviatori[1].cntrlChiudi := FALSE;
        deviatori[1].color:=USINT#0; //colre magazzino feed (da aggiornare con TUTTI i colori che non sono appartenenti ad un magazzino colore)

        magazzini[1].ID:=nastri[1].ID;
        magazzini[1].acceptedColor := USINT#0; // impostare colore
        magazzini[1].actualState := stato#stop;
        magazzini[1].CntrlForward := FALSE;
        magazzini[1].CntrlBackward := FALSE;
        magazzini[1].isForward := FALSE;
        magazzini[1].isBackward := FALSE;

        magazzini[1].maxCapacity := Capacity; // impostare capacità desiderata
        magazzini[1].currentStockLevel:=0;
        magazzini[1].StockisFull := FALSE;
        magazzini[1].currentMode := Tipi.InventoryMode#Fill; // di default vogliamo riempire i magazzini

        //coda
        nastri[n_mag].ID := n_mag;
        nastri[n_mag].colore := USINT#0;
        nastri[n_mag].actualState := stato#stop;
        nastri[n_mag].CntrlForward := FALSE;
        nastri[n_mag].CntrlBackward := FALSE;
        nastri[n_mag].isForward := FALSE;
        nastri[n_mag].isBackward := FALSE;

        deviatori[n_mag].ID:=nastri[n_mag].ID;
        deviatori[n_mag].sensore := FALSE;
        deviatori[n_mag].chiuso := FALSE;
        deviatori[n_mag].cntrlApri := FALSE;
        deviatori[n_mag].cntrlChiudi := FALSE;
        deviatori[n_mag].color:=USINT#0;

        magazzini[n_mag].ID:=nastri[n_mag].ID;
        magazzini[n_mag].acceptedColor := USINT#0; // impostare colore
        magazzini[n_mag].actualState := stato#stop;
        magazzini[n_mag].CntrlForward := FALSE;
        magazzini[n_mag].CntrlBackward := FALSE;
        magazzini[n_mag].isForward := FALSE;
        magazzini[n_mag].isBackward := FALSE;

        magazzini[n_mag].maxCapacity := Capacity; // impostare capacità desiderata
        magazzini[n_mag].currentStockLevel:=0;
        magazzini[n_mag].StockisFull := FALSE;
        magazzini[n_mag].currentMode := Tipi.InventoryMode#Fill; // di default vogliamo riempire i magazzini

        //secondo
        nastri[2].ID := 2;
        nastri[2].colore := USINT#1;
        nastri[2].actualState := stato#stop;
        nastri[2].CntrlForward := FALSE;
        nastri[2].CntrlBackward := FALSE;
        nastri[2].isForward := FALSE;
        nastri[2].isBackward := FALSE;

        deviatori[2].ID:=nastri[2].ID;
        deviatori[2].sensore := FALSE;
        deviatori[2].chiuso := FALSE;
        deviatori[2].cntrlApri := FALSE;
        deviatori[2].cntrlChiudi := FALSE;
        deviatori[2].color:=USINT#1;

        magazzini[2].ID:=nastri[2].ID;
        magazzini[2].acceptedColor := USINT#1; // impostare colore
        magazzini[2].actualState := stato#stop;
        magazzini[2].CntrlForward := FALSE;
        magazzini[2].CntrlBackward := FALSE;
        magazzini[2].isForward := FALSE;
        magazzini[2].isBackward := FALSE;

        magazzini[2].maxCapacity := Capacity; // impostare capacità desiderata
        magazzini[2].currentStockLevel:=0;
        magazzini[2].StockisFull := FALSE;
        magazzini[2].currentMode := Tipi.InventoryMode#Fill; // di default vogliamo riempire i magazzini

        //terzo
        nastri[3].ID := 3;
        nastri[3].colore := USINT#2;
        nastri[3].actualState := stato#stop;
        nastri[3].CntrlForward := FALSE;
        nastri[3].CntrlBackward := FALSE;
        nastri[3].isForward := FALSE;
        nastri[3].isBackward := FALSE;

        deviatori[3].ID:=nastri[3].ID;
        deviatori[3].sensore := FALSE;
        deviatori[3].chiuso := FALSE;
        deviatori[3].cntrlApri := FALSE;
        deviatori[3].cntrlChiudi := FALSE;
        deviatori[3].color:=USINT#2;

        magazzini[3].ID:=nastri[3].ID;
        magazzini[3].acceptedColor := USINT#2; // impostare colore
        magazzini[3].actualState := stato#stop;
        magazzini[3].CntrlForward := FALSE;
        magazzini[3].CntrlBackward := FALSE;
        magazzini[3].isForward := FALSE;
        magazzini[3].isBackward := FALSE;

        magazzini[3].maxCapacity := Capacity; // impostare capacità desiderata
        magazzini[3].currentStockLevel:=0;
        magazzini[3].StockisFull := FALSE;
        magazzini[3].currentMode := Tipi.InventoryMode#Fill; // di default vogliamo riempire i magazzini

        //quarto o ricetta
        nastri[4].ID := 4;
        nastri[4].colore := USINT#3;
        nastri[4].actualState := stato#stop;
        nastri[4].CntrlForward := FALSE;
        nastri[4].CntrlBackward := FALSE;
        nastri[4].isForward := FALSE;
        nastri[4].isBackward := FALSE;

        deviatori[4].ID:=nastri[4].ID;
        deviatori[4].sensore := FALSE;
        deviatori[4].chiuso := FALSE;
        deviatori[4].cntrlApri := FALSE;
        deviatori[4].cntrlChiudi := FALSE;
        deviatori[4].color:=USINT#3;

        magazzini[4].ID:=nastri[4].ID;
        magazzini[4].acceptedColor := USINT#3; // impostare colore
        magazzini[4].actualState := stato#stop;
        magazzini[4].CntrlForward := FALSE;
        magazzini[4].CntrlBackward := FALSE;
        magazzini[4].isForward := FALSE;
        magazzini[4].isBackward := FALSE;

        magazzini[4].maxCapacity := Capacity; // impostare capacità desiderata
        magazzini[4].currentStockLevel:=0;
        magazzini[4].StockisFull := FALSE;
        magazzini[4].currentMode := Tipi.InventoryMode#Fill; // di default vogliamo riempire i magazzini

END_PROGRAM

(* ---- MainProgram.st ---- *)
USING tipi;
USING Libreria;

PROGRAM MainProgram

    VAR
        tStopMotor : INT:=5;//tempo movimento motori
        n_pacchi :INT:=10;
        n_mag : INT:=3;// numero magazzini

        nastri : ARRAY[1..3] OF nastro;
        deviatori : ARRAY[1..3] OF deviatore;
        magazzini : ARRAY[1..3+1] OF magazzino;

        fineProcesso: BOOL := FALSE;
        tempotrascorso: BOOL := FALSE;
        flag : BOOL:=FALSE;
    END_VAR

    VAR_TEMP
        i:INT;
    END_VAR

    FOR i:=1 TO n_mag DO //inizializzare componenti
        nastri[i].Init(i);
        deviatori[i].Init(i);
        magazzini[i].Init(i);
    END_FOR;

    magazzini[n_mag+1].Init(n_mag+1);

    IF not(n_pacchi>0) THEN //se non ci sono pacchi fine smistamento
        fineProcesso:= TRUE;
    END_IF;

    WHILE NOT(fineProcesso) DO //finche ci sono pacchi da smistare
        i:=1;
        Flag := FALSE;

        IF n_pacchi = 0 THEN
            fineProcesso := TRUE;
        END_IF;

        WHILE i<n_mag+1 DO

            nastri[i].CntrlForward := TRUE;//movimento avanti motore nastro
            nastri[i].isEmpty() := FALSE;// fotocellula con pacchi
            nastri[i].Update();//aggiorna stato nastro

            if i>1 THEN
                deviatori[i-1].sensore_presenza := FALSE; //spegni il sensore del deviatore precendente
            END_IF;

            tempotrascorso := Timer(tStopMotor);
            deviatori[i].sensore_presenza := TRUE;//il deviatore vede un pacco
            deviatori[i].smista:=TRUE;// controllato se il pacco è da smistare

            IF tempotrascorso AND deviatori[i].sensore_presenza THEN // controlla se il sensore vede il pacco dopo il movimento del motore
                nastri[i].CntrlForward := FALSE;//spegni motore
                nastri[i].update();//aggiorna stato nastro

                IF NOT(magazzini[i].isFull) AND deviatori[i].smista THEN //controlla che il magazzino sia libero, il colore del pacco corrisponde con il colore del magazzino
                    deviatori[i].devia();// devia il pacco
                    magazzini[i].CntrlForward := TRUE;//attiva motore magazzino
                    magazzini[i].update();//aggiorna lo stato del nastro magazzino
                    nastri[i].isEmpty() := TRUE;//spegne la fotocellula nastro
                    deviatori[i].sensore_presenza := FALSE;// spegne sensore presenza pacco
                    magazzini[i].fotocellula := TRUE;// la fotocellula del magazzino vede il pacco

                    tempotrascorso := Timer(tStopMotor);
                    magazzini[i].fotocellula := FALSE;// la fotocellula non vede più il pacco che è entrato a magazzino

                    n_pacchi := n_pacchi-1; //il numero di pacchi cala
                    magazzini[i].spazio := magazzini[i].spazio - 1; //lo spazio del magazzino cala

                    IF magazzini[i].spazio = 0 THEN//se non c'è più spazio il magazzino diventa pieno
                        magazzini[i].isFull:=TRUE;
                    END_IF;

                    flag:=TRUE;// flag per segnare che i pacchi sono già stati ridotti
                    i:=n_mag;

                END_IF;

            END_IF;

            i:=i+1;

        END_WHILE;

        IF i=n_mag+1 AND NOT(Flag) THEN //se abbiamo passato tutti i magazzini e i pacchi non sono stati ridotti entra nel magazzino scarto finale
            n_pacchi:= n_pacchi-1; //il numero di pacchi cala
            magazzini[n_mag+1].spazio := magazzini[n_mag].spazio - 1;  //lo spazio del magazzino scarto finale cala
            IF magazzini[n_mag+1].spazio = -1 THEN // se lo spazio del magazzino finale da 0 passa a -1 significa che vogliamo forzare un pacco che non è stato smistato nel magazzino finale pieno
                fineProcesso := TRUE; //esci dal ciclo perche non posso più carica
            END_IF;
        END_IF;

    END_WHILE;

    //smistamento completato

END_PROGRAM
